TYPE IoC13336Mppc :
STRUCT	
	(** One relay manage 2 MPPCs -> The wide MPPC output is physically and only connected. It also manages the relay of the Narrow MPPC output **)
	OutputMppcRelayPower : BOOL; 
END_STRUCT
END_TYPE

(* stored: Version 1.1.0.1, ProductVersion 3.1.4024.3
   DUT IoC13336Mppc: Id {ac6760c8-98f7-47ec-ae96-9e57b8dd4f17} *)
